# EPICS substitutions: streamApp/pluginDb/cross.substitutions
# cross.substitutions

file cross.template
{
    pattern
    {   N,  P,          R    }
    {   1,  "\$(CAM)",  ":"  }
    {   2,  "\$(CAM)",  ":"  }
    {   3,  "\$(CAM)",  ":"  }
    {   4,  "\$(CAM)",  ":"  }
}

file crossLimits.template
{
	{
		P		= "\$(CAM)",
		R		= ":",
	}
}
